// TIA Portal V18 export
FUNCTION_BLOCK "FB_PT_Motors"   // FB2, LAD
{ S7_Optimized_Access := 'TRUE' }
// stored: MemoryReserve 100, SetENOAutomatically false
BEGIN

REGION Network 1: Motor_1
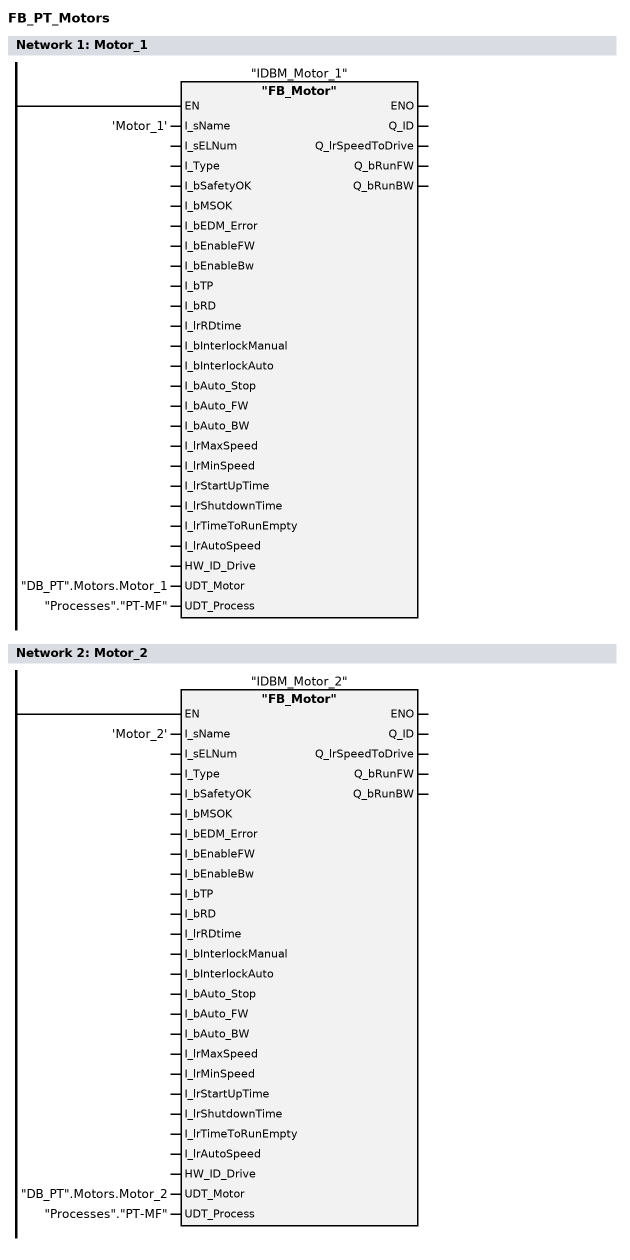
   RUNG wire#powerrail
      "IDBM_Motor_1"(I_sName := 'Motor_1', I_sELNum :=, I_Type :=, I_bSafetyOK :=, I_bMSOK :=, I_bEDM_Error :=, I_bEnableFW :=, I_bEnableBw :=, I_bTP :=, I_bRD :=, I_lrRDtime :=, I_bInterlockManual :=, I_bInterlockAuto :=, I_bAuto_Stop :=, I_bAuto_FW :=, I_bAuto_BW :=, I_lrMaxSpeed :=, I_lrMinSpeed :=, I_lrStartUpTime :=, I_lrShutdownTime :=, I_lrTimeToRunEmpty :=, I_lrAutoSpeed :=, HW_ID_Drive :=, UDT_Motor := "DB_PT".Motors.Motor_1, UDT_Process := "Processes"."PT-MF", Q_ID =>, Q_lrSpeedToDrive =>, Q_bRunFW =>, Q_bRunBW =>)
   END_RUNG
   // the same network as SCL:
   "IDBM_Motor_1"(I_sName := 'Motor_1', UDT_Motor := "DB_PT".Motors.Motor_1, UDT_Process := "Processes"."PT-MF");   // "FB_Motor"
END_REGION

REGION Network 2: Motor_2
   RUNG wire#powerrail
      "IDBM_Motor_2"(I_sName := 'Motor_2', I_sELNum :=, I_Type :=, I_bSafetyOK :=, I_bMSOK :=, I_bEDM_Error :=, I_bEnableFW :=, I_bEnableBw :=, I_bTP :=, I_bRD :=, I_lrRDtime :=, I_bInterlockManual :=, I_bInterlockAuto :=, I_bAuto_Stop :=, I_bAuto_FW :=, I_bAuto_BW :=, I_lrMaxSpeed :=, I_lrMinSpeed :=, I_lrStartUpTime :=, I_lrShutdownTime :=, I_lrTimeToRunEmpty :=, I_lrAutoSpeed :=, HW_ID_Drive :=, UDT_Motor := "DB_PT".Motors.Motor_2, UDT_Process := "Processes"."PT-MF", Q_ID =>, Q_lrSpeedToDrive =>, Q_bRunFW =>, Q_bRunBW =>)
   END_RUNG
   // the same network as SCL:
   "IDBM_Motor_2"(I_sName := 'Motor_2', UDT_Motor := "DB_PT".Motors.Motor_2, UDT_Process := "Processes"."PT-MF");   // "FB_Motor"
END_REGION
END_FUNCTION_BLOCK
